// TIA Portal project "FicherTechnik_V1" (V16)

(* hardware
DEVICE "S7-1200 station_1"  S7-1200 Station
   slot 0: "Rack_0"  S7-1200 Rack  Rack  V1.0
   slot 1: "PLC_1"  CPU 1214C DC/DC/DC  6ES7 214-1AG40-0XB0  V4.4
*)

// ===== PLC "PLC_1"  CPU 1214C DC/DC/DC =====

VAR_GLOBAL   // PLC tag table "Default tag table"
   "magazineFilled" AT %I0.0 : Bool;
   "turntableInHomePosition" AT %I0.1 : Bool;
   "transferUnitReady" AT %I0.2 : Bool;
   "transferReadyLED" AT %Q0.0 : Bool;
   "turntableMotor" AT %Q0.1 : Bool;
   "drillingMotor" AT %Q0.2 : Bool;
   "weldingLight" AT %Q0.3 : Bool;
   "magazinePusher" AT %Q0.4 : Bool;
END_VAR

DATA_BLOCK "DB_Workpieces"   // DB1
{ S7_Optimized_Access := 'TRUE' }
VERSION : 0.1
   VAR
      magazinePart : Bool;
      drillingRawPart : Bool;
      drillingFinishedPart : Bool;
      weldingRawPart : Bool;
      weldingFinishedPart : Bool;
      transferPart : Bool;
      S4_Lastscan : Bool;
      pushActive : Bool;
      TRANSFER_PART_READY : Int := 1;
      TRANSFER_PART_DONE : Int := 2;
      TRANSFER_PART_IDLE : Int := 0;
   END_VAR
BEGIN
END_DATA_BLOCK

DATA_BLOCK "MagazineManager_DB"   // DB2
{ S7_Optimized_Access := 'TRUE' }
VERSION : 0.1
// stored: InstanceOfName MagazineManager
"MagazineManager"
BEGIN
END_DATA_BLOCK

DATA_BLOCK "DrillingManager_DB"   // DB3
{ S7_Optimized_Access := 'TRUE' }
VERSION : 0.1
// stored: InstanceOfName DrillingManager
"DrillingManager"
BEGIN
END_DATA_BLOCK

DATA_BLOCK "WeldingManager_DB"   // DB4
{ S7_Optimized_Access := 'TRUE' }
VERSION : 0.1
// stored: InstanceOfName WeldingManager
"WeldingManager"
BEGIN
END_DATA_BLOCK

DATA_BLOCK "Modbus_TCP_DB"   // DB6
{ S7_Optimized_Access := 'TRUE' }
VERSION : 0.1
   VAR
      HandshakeReg : Int;   // Buffer for read /write
      ConnParams : TCON_IP_v4;
      ReqTrigger : Bool;   // Fires one request
      ModeSelect : USInt;   // Client Mode selector: 0=Read, 1=Write
      Done : Bool;
      Busy : Bool;
      Error : Bool;
      Status : Word;
   END_VAR
BEGIN
   ConnParams.RemoteAddress.ADDR[1] := 192;
   ConnParams.RemoteAddress.ADDR[2] := 168;
   ConnParams.RemoteAddress.ADDR[3] := 50;
   ConnParams.RemoteAddress.ADDR[4] := 20;
   ConnParams.RemotePort := 502;
   ConnParams.LocalPort := 0;
   ConnParams.InterfaceId := 64;
   ConnParams.ID := 1;
   ConnParams.ConnectionType := 11;
   ConnParams.ActiveEstablished := TRUE;
END_DATA_BLOCK

DATA_BLOCK "ModbusManager_DB"   // DB7
{ S7_Optimized_Access := 'TRUE' }
VERSION : 0.1
// stored: InstanceOfName ModbusManager
"ModbusManager"
BEGIN
END_DATA_BLOCK

DATA_BLOCK "DB_OPCUA_Interface"   // DB8
{ S7_Optimized_Access := 'TRUE' }
VERSION : 0.1
   VAR
      Turntable : Struct
         inPosition : Bool;
         magazineEmpty : Bool;
         motorTurntable : Bool;
         drillActive : Bool;
         weldActive : Bool;
         magazinePart : Bool;
         transferReady : Bool;
         sliderMagazine : Bool;
         weldingPart : Bool;
         drillPart : Bool;
      END_STRUCT;
      Commands : Struct
         startCommand : Bool := true;
         stopCommand : Bool := false;
         resetCommand : Bool;
      END_STRUCT;
      Diagnostics : Struct
         completed_pieces : DInt;
         peerCommunicationOK : Bool;
         controllerActive : Bool;
      END_STRUCT;
   END_VAR
BEGIN
END_DATA_BLOCK

FUNCTION_BLOCK "DrillingManager"   // FB1, SCL
{ S7_Optimized_Access := 'TRUE' }
VERSION : 0.1
   VAR
      drillingConditionMet : Bool;
      drillingTimer : IEC_TIMER;
   END_VAR
BEGIN
   (*
           The purpose of this FB is to control the logic and timings of the the drilling motor(Q9) at station 2.
           The drilling is run for three seconds when the raw part is present.
           The transition from drillingRawPart -> drillingFinishedPart is made upon completion.
       *)

   (*
       Conditions to start drilling:
           1. Raw(undrilled) part is in station 2: drillingRawPart = TRUE;
           2. Turntable is in position: tableInHomePosition = TRUE
           3. Turntable not rotating: turntableMotor = FALSE
   *)

   #drillingConditionMet := "DB_Workpieces".drillingRawPart
   AND (NOT "turntableMotor")
   AND "turntableInHomePosition";

   (*
       If the drilling conditions are met, start the timer for 3 seconds
   *)
   #drillingTimer.TON(IN := #drillingConditionMet,
   PT := T#3s
   );

   (*
       For as long as drillingTimer is ticking,m drive the drilling motor
   *)

   "drillingMotor" := (#drillingTimer.IN AND NOT #drillingTimer.Q);

   (*
       Transition Flags upon completion:
       When the timer elapses:
           - Clear "drillingRawPart",
           - Set "drillingFinishedPart"
   *)
   IF #drillingTimer.Q THEN
       "DB_Workpieces".drillingRawPart := FALSE;
       "DB_Workpieces".drillingFinishedPart := TRUE;
   END_IF;
END_FUNCTION_BLOCK

FUNCTION_BLOCK "MagazineManager"   // FB2, SCL
{ S7_Optimized_Access := 'TRUE' }
VERSION : 0.1
   VAR
      sliderConditionMet : Bool;
      magazineTimer : IEC_TIMER;
   END_VAR
BEGIN
   (*\
        The purpose of this function block is to control the magazine slider (actuated via Q7 which o).
        One workpiece is pushed from the magazine into the turntable nest at station 1, if slideConditinMet,
        and outputs True. ( must be wired to magazinePart).
       *)

   (*
       Conditions to Push:
           1. Magazine is not empty. (magazineFilled = TRUE)
           2. Nest at station 1 is empty: DB_Workpieces.magazinePart = FALSE
           3. Turntable is in position: tableInHomePosition = TRUE
           4. The motor is not rotating: turntableMotor = FALSE
   *)

   #sliderConditionMet := (NOT "magazineFilled")
   AND (NOT "DB_Workpieces".magazinePart)
   AND "turntableInHomePosition"
   AND (NOT "turntableMotor");

   (*
       Because need  not to use the sliderConditionMet as the holding condition of the timer, 
       becuase it can chane 1 ms later, even before the piece has been pushed into the timer( timer doesn't even start)

       we use it only to set the pushActive flag, which is the one that controls the state
   *)
   IF #sliderConditionMet AND NOT "DB_Workpieces".magazinePart THEN
       "DB_Workpieces".pushActive := TRUE;
   END_IF;
   (*
       Based on the Time IN and Timer out, we control the slider activation duration.
       The TON timer is gateed by the sliderConditionMet.
       While Timer_IN = TRUE, the timer counts up. When ET>PT, Q = TREU.
       Once conditions are no longer met ( magazinePart set), IN drops and timer resets automatically in the next scan.
   *)

   #magazineTimer.TON(IN := "DB_Workpieces".pushActive,
   PT := T#1500ms);

   (*
       Drive the Slider Output.
       Q7 (magazinePusher) get actuated while the time is still on and running.
       magazineTimer.In going true means we are in push phase
       The spring returns the slider automatically, when magazinePusher de-enegizes
   *)
   "magazinePusher" := #magazineTimer.IN AND (NOT #magazineTimer.Q);

   (*
       Set magazinePart FLAG.
       when the timer elapses (Q = TRUE), the workpiece is confirmed in the nest.
       Set the flaf so that the system knows station 1 is occupied. 
       This also prevents re-pushing in the next scan cycle.
   *)
   IF #magazineTimer.Q THEN
       "DB_Workpieces".magazinePart := TRUE;
       "DB_Workpieces".pushActive := FALSE;
   END_IF;
END_FUNCTION_BLOCK

FUNCTION_BLOCK "WeldingManager"   // FB3, SCL
{ S7_Optimized_Access := 'TRUE' }
VERSION : 0.1
   VAR
      weldingConditionMet : Bool;
      weldingTimer : IEC_TIMER;
   END_VAR
BEGIN
   (*
         Purpose: To control and monitor the welding station of the sytem. This FB is responsible for starting, and stopping the welding process.

         A part is welded fro 5 seconds (as per the documentation), when welding is done, the FB transitions from
         weldingRawPart -> weldingFinishedPart.
       *)

   (*
       Welding Start Conditions:
           Raw (pre-welded) part is present i station 3: weldingRawPart = TRUE;
           Turntable is in Position: turntableInHomePosition = TRUE;
           Turntable is not rotating. turntableMotor = FALSE
   *)
   #weldingConditionMet := "DB_Workpieces".weldingRawPart AND (NOT "turntableMotor") AND "turntableInHomePosition";

   (*
       If the conditions are met, start the welding timer
   *)
   #weldingTimer.TON(IN := #weldingConditionMet,
   PT:= T#5S
   );

   (*
       As long as the timer is ticking, weld the part
   *)
   "weldingLight" := #weldingTimer.IN AND (NOT #weldingTimer.Q); //timer started, but has not finished yet.

   (*
       Upon completion, transition the flags:
           - Clear weldingRawPart
           -Set weldingFinishedPart
   *)
   IF #weldingTimer.Q THEN
       "DB_Workpieces".weldingFinishedPart := TRUE;
       "DB_Workpieces".weldingRawPart := FALSE;
   END_IF;
END_FUNCTION_BLOCK

FUNCTION_BLOCK "ModbusManager"   // FB4, SCL
{ S7_Optimized_Access := 'TRUE' }
VERSION : 0.1
   VAR
      State : Int;   // 0=Read, 1=WaitRead, 2=Eval, 3=Write. 4=WaitWrite
      WriteVal : Int;
      Static_1 : IEC_TIMER;
      Static_2 : IEC_TIMER;
      waitingAck : Bool;
   END_VAR
BEGIN
   (*
   Decription: This following function block implements the handshake between Siemens and Allen Bradley. When the transferPart =True, Siemens 
   need to notify the Allen Bradley by sending "TransferReady Packet over the network.

   *)

   CASE #State OF
       0: //Trigger Read
           IF NOT "Modbus_TCP_DB".Busy THEN
               "Modbus_TCP_DB".ModeSelect := 0; //SET THE MODE TO READ
               "Modbus_TCP_DB".ReqTrigger := TRUE; //Trigger Read
               #State := 1; //Transition into WaitRead state
           END_IF;
       1: //Waiting for Read to complete.
           IF "Modbus_TCP_DB".Busy OR "Modbus_TCP_DB".Done THEN
               "Modbus_TCP_DB".ReqTrigger := FALSE; //Reset trigger
           END_IF;

           IF "Modbus_TCP_DB".Done THEN

               #State := 2; // transition into Evaluation State.
           ELSIF "Modbus_TCP_DB".Error THEN
               #State := 0; //If error occured during read, set the state to 0.
           END_IF;
       2: //Evaluation state
           IF "Modbus_TCP_DB".HandshakeReg = "DB_Workpieces".TRANSFER_PART_DONE THEN
               // if Allen Bradley is done, we acknowledge with 0, and then release the Siemens to proceed.
               #WriteVal := "DB_Workpieces".TRANSFER_PART_IDLE;
               "DB_Workpieces".transferPart := FALSE;
               #waitingAck := FALSE;
               "DB_OPCUA_Interface".Diagnostics.completed_pieces := "DB_OPCUA_Interface".Diagnostics.completed_pieces + 1;
               #State := 3;
           ELSIF "Modbus_TCP_DB".HandshakeReg = "DB_Workpieces".TRANSFER_PART_IDLE AND
               "DB_Workpieces".transferPart AND NOT #waitingAck THEN
               // Transfer part is ready -> signal the AB
               #WriteVal := "DB_Workpieces".TRANSFER_PART_READY;
               #waitingAck := TRUE;
               #State := 3;
           ELSE
               #State := 0; // Do Nothing and skeep pooling
           END_IF;
       3: //Trigger Write
           IF NOT "Modbus_TCP_DB".Busy THEN
               "Modbus_TCP_DB".HandshakeReg := #WriteVal;
               "Modbus_TCP_DB".ModeSelect := 1; // SET THE MODE TO WRITE.
               "Modbus_TCP_DB".ReqTrigger := TRUE;
               #State := 4; //SET THE state to Wait for Write.
           END_IF;
       4: //WAIT FOR WRITE TO COMPLETE.
           "Modbus_TCP_DB".ReqTrigger := FALSE;

           IF "Modbus_TCP_DB".Done THEN
               #State := 0;
           ELSIF "Modbus_TCP_DB".Error THEN
               #State := 0; //Re-try from READ.
           END_IF;
   END_CASE;
END_FUNCTION_BLOCK

FUNCTION "TurnTableControl" : Void   // FC1, SCL
{ S7_Optimized_Access := 'TRUE' }
VERSION : 0.1
   VAR_TEMP
      rotationPermitted : Bool;
      rotationBlocked : Bool;
   END_VAR
BEGIN
   (*
       Description: This is a Function(FC not funcion block) that runs every scan to decide whether turntable motor should run.
                    It implements both the PERMISSION Logic ( why the table CAN rotate), and the INTERLOCK logic ( whyy the turntable MUST NOT rotate).
                    Since this is a pure conbinational logic, and not timiers are not needed, it is defined as a Function as opposed to Function Block .
       *)

   (*
       ============================================================================================================
       ROTATION PERMISION
       ============================================================================================================

       The Table is allowed to rotate if and only if at least on of the the following is TRUE:
           1. magazinePart = TRUE.
           2. drillingFinishedPart = TRUE
           3. weldingFinishedPart = TRUE
       These are OR'ed torgther and any one fo them uis sufficient to permit rotation
       Note: drillingRawPart and WeldingRawPart do not permit rotation because a raw part means processing is in progress opr is still needed. the table must wait .
   *)

   #rotationPermitted := "DB_Workpieces".magazinePart OR "DB_Workpieces".drillingFinishedPart OR "DB_Workpieces".weldingFinishedPart;

   (*
       table will not move until transferPart is set to False. We must thus check the status of "Modbus_DB,"HoldingRegister[0], to see if 
       Allen-Bradley has written TRANSFER_PART_DONE code to this, if so, we set "DB_Workpieces".trasnsferPart = FALSE, and immediately, set
       "Modbus_DB,"HoldingRegister[0] to TRANSFER_PART_IDLE
   *)
   //IF "ModbusTCP_DB".HoldingRegister[0] = "DB_Workpieces".TRANSFER_PART_DONE THEN
       //"DB_Workpieces".transferPart := FALSE;
       //"ModbusTCP_DB".HoldingRegister[0] := "DB_Workpieces".TRANSFER_PART_IDLE;
       //"transferReadyLED" := FALSE;
   //END_IF;

   (*
       =============================================================
       ROTATION BLOCKING
       =============================================================
       The table is BLOCKED from rotating if ANY of the following is TRUE:
           1. transferPart = TRUE: a finished workpiece is in station 4, the table must not move until the piece is picked up by the other PLC., and resets this flag.
           2. drillingRawPart = TRUE:
               Station 2 has an undrilled workpiece. Either drilling is in progress or has not started yet.
           3. weldingRawPart = True:
               Same as station 2, if station 3 has un-welded, drilled workpiece, or welding is in progress, the table must not move at all.
           4. magazinePusher = true (Q7 excited):
                If magazine slider in extended into the turntable nest zone, the table must not move. ( this would cause machanical collision, and damage the model).
           5. S2 is true:
               The transfer unit is in the turntable direction, too far that is actuated S2.
   These conditions are also OR'ed to build rotation blocked flag
   *)

   #rotationBlocked :=
   "DB_Workpieces".transferPart
   OR "DB_Workpieces".drillingRawPart
   OR "DB_Workpieces".weldingRawPart
   OR "transferUnitReady";
   //OR "transferReadyLED";

   (*
       Turn the Motor when all of the following are True:
           1. rotationPermitted = True
           2. rotationBlocked = False ( No interlocking)
           3. Turntable is currently is position (S4 = TRUE) or the motor has been turning ( self-sustained latching)
   *)


   "turntableMotor" := (#rotationPermitted AND NOT #rotationBlocked) AND ("turntableInHomePosition" OR "turntableMotor");
END_FUNCTION

FUNCTION "RotateWorkpieces" : Void   // FC2, SCL
{ S7_Optimized_Access := 'TRUE' }
VERSION : 0.1
   VAR_TEMP
      S4_RisingEdge : Bool;
   END_VAR
BEGIN
   (*
           This detects the rising edge of turntableInHomePosition(S4), and shifts the workpieces by one station around the table.

           This must be called every scan, and must be the first block called from the main OB.
           Note: Rising edge is implemented manually using S4_Lastscan stored in DB_Workpieces. This is because FC block do not have static variables
       *)

   (*
       Step 1: Detect Rising Edge of S4(tableInHomePosition):

       S4 is normally-open limit switch that fires when the turntable nest is aligned with all stations.
       We only need only one FIRST Scan where it becomes true to trigger for a single data rotation.

       S4_Lastscan holds the value of S4 from the previous PLC scan cycle ( stored in global DB so that is persistent across scans)
   *)
   #S4_RisingEdge := "turntableInHomePosition" AND (NOT "DB_Workpieces".S4_Lastscan);

   //update the S4_Lastscan for the next cycle
   "DB_Workpieces".S4_Lastscan := "turntableInHomePosition";

   (* Step 2: Rotate Workpieces(if rising edge detected):
       If Rising Edge is detected, rotate the workpieces data
       Each workpiece has physically moved 90 degrees clockwise: 1->2->3->4->1. 
       we need to mirror this in software by shifting the flags forward one station.

       The following is rotation chain ( executed in reverse order):
            weldingFinishedPart -> transferPart
            drillingFinishedPart -> weldingRawPart
            magazinePart -> drillingRawPart
            station 4 -> station 1: ( transferPart clears, picked up by the other PLC).
            magazinePart clears after rotation
   *)

   IF #S4_RisingEdge THEN
       //Strep 2.1: Finished part from station 3 advances to station 4(handover) or transfer
       "DB_Workpieces".transferPart := "DB_Workpieces".weldingFinishedPart;

       //Step 2.2: Drilled Part from Station 2 moves to Station 3
       "DB_Workpieces".weldingRawPart := "DB_Workpieces".drillingFinishedPart;

       //Step 2.3: New Raw part from station 1 moves to Station 2
       "DB_Workpieces".drillingRawPart := "DB_Workpieces".magazinePart;

       //step 2.4: After rotating parts, clear source flags
       "DB_Workpieces".weldingFinishedPart := FALSE;
       "DB_Workpieces".drillingFinishedPart := FALSE;
       "DB_Workpieces".magazinePart := FALSE;
       //if A part is Ready
       //IF "DB_Workpieces".transferPart THEN
       // "ModbusTCP_DB".HoldingRegister[0] := "DB_Workpieces".TRANSFER_PART_READY;
       // "transferReadyLED" := TRUE;
       // END_IF;

   END_IF;


   //Siemen's Active Light
   IF "DB_Workpieces".magazinePart OR
       "DB_Workpieces".drillingRawPart OR
       "DB_Workpieces".weldingRawPart OR
       NOT "turntableInHomePosition" OR
       "magazinePusher" THEN
       "transferReadyLED" := TRUE;
   ELSE
       "transferReadyLED" := FALSE;
   END_IF;
END_FUNCTION

FUNCTION "OPCServerManager" : Void   // FC3, SCL
{ S7_Optimized_Access := 'TRUE' }
VERSION : 0.1
BEGIN
   "DB_OPCUA_Interface".Turntable.drillActive := "drillingMotor";
   "DB_OPCUA_Interface".Turntable.weldActive := "weldingLight";
   "DB_OPCUA_Interface".Turntable.inPosition := "turntableInHomePosition";
   "DB_OPCUA_Interface".Turntable.magazineEmpty := "magazineFilled";
   "DB_OPCUA_Interface".Turntable.magazinePart := "DB_Workpieces".magazinePart;
   "DB_OPCUA_Interface".Turntable.transferReady := "DB_Workpieces".transferPart;
   "DB_OPCUA_Interface".Turntable.magazinePart := "DB_Workpieces".magazinePart;
   "DB_OPCUA_Interface".Turntable.drillPart := "DB_Workpieces".drillingRawPart;
   "DB_OPCUA_Interface".Turntable.sliderMagazine := "magazinePusher";
   "DB_OPCUA_Interface".Turntable.motorTurntable := "turntableMotor";

   "DB_OPCUA_Interface".Diagnostics.controllerActive := "transferReadyLED";
   "DB_OPCUA_Interface".Diagnostics.peerCommunicationOK := NOT "Modbus_TCP_DB".Error;
END_FUNCTION

ORGANIZATION_BLOCK "Main"   // OB1, LAD, ProgramCycle
TITLE = "Main Program Sweep (Cycle)"
{ S7_Optimized_Access := 'TRUE' }
VERSION : 0.1
   VAR_INPUT
      Initial_Call : Bool;   // Initial call of this OB
      Remanence : Bool;   // =True, if remanent data are available
   END_VAR
BEGIN

REGION Network 1
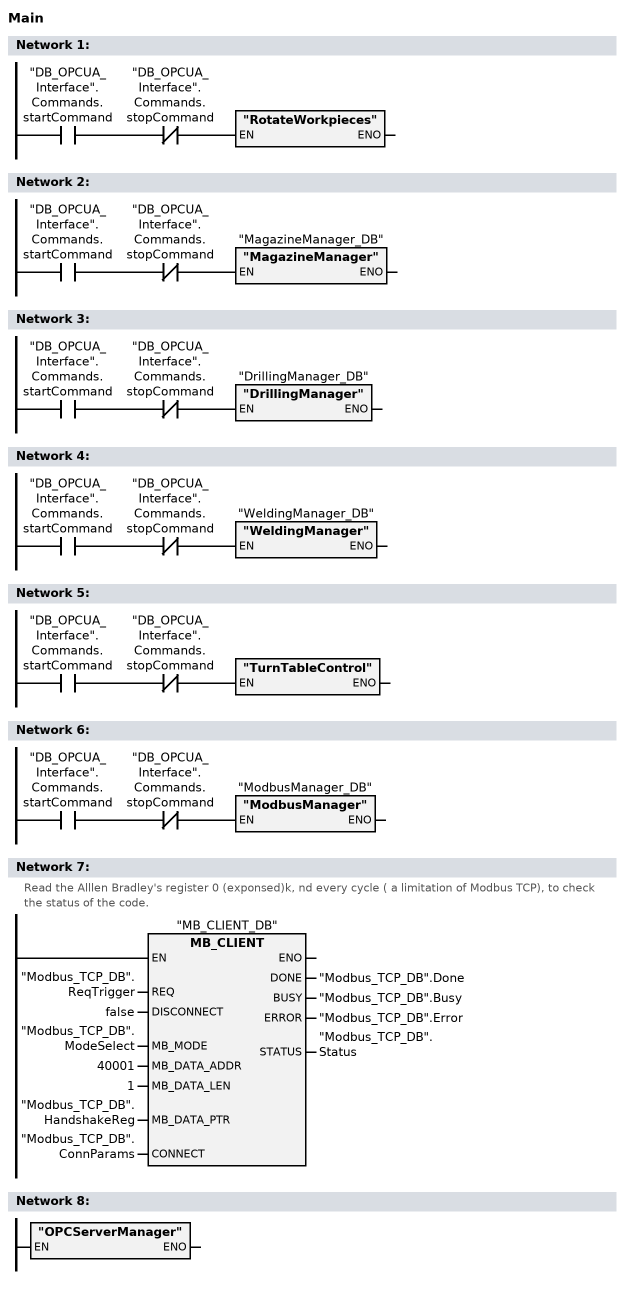
   RUNG wire#powerrail
      Contact( "DB_OPCUA_Interface".Commands.startCommand )
      I_Contact( "DB_OPCUA_Interface".Commands.stopCommand )
      "RotateWorkpieces"()
   END_RUNG
   // the same network as SCL:
   IF "DB_OPCUA_Interface".Commands.startCommand AND NOT "DB_OPCUA_Interface".Commands.stopCommand THEN
       "RotateWorkpieces"();
   END_IF;
END_REGION

REGION Network 2
   RUNG wire#powerrail
      Contact( "DB_OPCUA_Interface".Commands.startCommand )
      I_Contact( "DB_OPCUA_Interface".Commands.stopCommand )
      "MagazineManager_DB"()
   END_RUNG
   // the same network as SCL:
   IF "DB_OPCUA_Interface".Commands.startCommand AND NOT "DB_OPCUA_Interface".Commands.stopCommand THEN
       "MagazineManager_DB"();   // "MagazineManager"
   END_IF;
END_REGION

REGION Network 3
   RUNG wire#powerrail
      Contact( "DB_OPCUA_Interface".Commands.startCommand )
      I_Contact( "DB_OPCUA_Interface".Commands.stopCommand )
      "DrillingManager_DB"()
   END_RUNG
   // the same network as SCL:
   IF "DB_OPCUA_Interface".Commands.startCommand AND NOT "DB_OPCUA_Interface".Commands.stopCommand THEN
       "DrillingManager_DB"();   // "DrillingManager"
   END_IF;
END_REGION

REGION Network 4
   RUNG wire#powerrail
      Contact( "DB_OPCUA_Interface".Commands.startCommand )
      I_Contact( "DB_OPCUA_Interface".Commands.stopCommand )
      "WeldingManager_DB"()
   END_RUNG
   // the same network as SCL:
   IF "DB_OPCUA_Interface".Commands.startCommand AND NOT "DB_OPCUA_Interface".Commands.stopCommand THEN
       "WeldingManager_DB"();   // "WeldingManager"
   END_IF;
END_REGION

REGION Network 5
   RUNG wire#powerrail
      Contact( "DB_OPCUA_Interface".Commands.startCommand )
      I_Contact( "DB_OPCUA_Interface".Commands.stopCommand )
      "TurnTableControl"()
   END_RUNG
   // the same network as SCL:
   IF "DB_OPCUA_Interface".Commands.startCommand AND NOT "DB_OPCUA_Interface".Commands.stopCommand THEN
       "TurnTableControl"();
   END_IF;
END_REGION

REGION Network 6
   RUNG wire#powerrail
      Contact( "DB_OPCUA_Interface".Commands.startCommand )
      I_Contact( "DB_OPCUA_Interface".Commands.stopCommand )
      "ModbusManager_DB"()
   END_RUNG
   // the same network as SCL:
   IF "DB_OPCUA_Interface".Commands.startCommand AND NOT "DB_OPCUA_Interface".Commands.stopCommand THEN
       "ModbusManager_DB"();   // "ModbusManager"
   END_IF;
END_REGION

REGION Network 7
   // Read the Alllen Bradley's register 0 (exponsed)k, nd every cycle ( a limitation of Modbus TCP), to check the status of the code.
   "MB_CLIENT_DB"(REQ := "Modbus_TCP_DB".ReqTrigger,   // MB_CLIENT
                  DISCONNECT := false,
                  MB_MODE := "Modbus_TCP_DB".ModeSelect,
                  MB_DATA_ADDR := 40001,
                  MB_DATA_LEN := 1,
                  MB_DATA_PTR := "Modbus_TCP_DB".HandshakeReg,
                  CONNECT := "Modbus_TCP_DB".ConnParams,
                  DONE => "Modbus_TCP_DB".Done,
                  BUSY => "Modbus_TCP_DB".Busy,
                  ERROR => "Modbus_TCP_DB".Error,
                  STATUS => "Modbus_TCP_DB".Status);
END_REGION

REGION Network 8
   RUNG wire#powerrail
      "OPCServerManager"()
   END_RUNG
   // the same network as SCL:
   "OPCServerManager"();
END_REGION
END_ORGANIZATION_BLOCK